FUNCTION_BLOCK c_bar_in (* Basic FB with empty ECC *)
  (* Standard: 61499-2 *)
  (* Version 1.0, 2020-08-20, Administrator *)
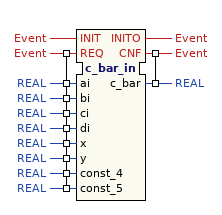
  EVENT_INPUT
    INIT;
    REQ WITH ai, bi, ci, x, di, y, const_5, const_4;
  END_EVENT
  EVENT_OUTPUT
    INITO;
    CNF WITH c_bar;
  END_EVENT
  VAR_INPUT
    ai : REAL;
    bi : REAL;
    ci : REAL;
    di : REAL;
    x : REAL;
    y : REAL;
    const_4 : REAL;
    const_5 : REAL;
  END_VAR
  VAR_OUTPUT
    c_bar : REAL;
  END_VAR
  VAR
    x2 : REAL; (* Internal Variable *)
    y2 : REAL; (* Internal Variable *)
    A : REAL; (* Internal Variable *)
    B : REAL; (* Internal Variable *)
    C : REAL; (* Internal Variable *)
  END_VAR
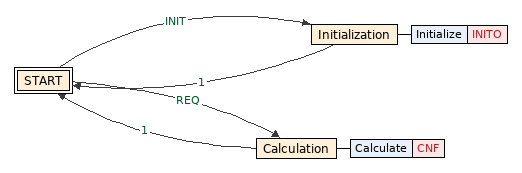
  EC_STATES
    START; (* Initial State *)
    Initialization : Initialize -> INITO;
    Calculation : Calculate -> CNF;
  END_STATES
  EC_TRANSITIONS
    START TO Initialization := INIT;
    Initialization TO START := 1;
    START TO Calculation := REQ;
    Calculation TO START := 1;
  END_TRANSITIONS
  ALGORITHM Initialize IN ST: (* New Algorithm *)

  END_ALGORITHM
  ALGORITHM Calculate IN ST: (* New Algorithm *)
//A
x2 := x*ai + y*ci;
y2 := x*bi + y*di;

A := x2*x + y2*y;

//B
B := const_4*x + const_5*y;

//C = -1

//
c_bar := A + B -1;
  END_ALGORITHM
END_FUNCTION_BLOCK
